PROGRAM EIP_COM
VAR
	eip_input AT%I* : ARRAY [0..63] OF BYTE;
	eip_output AT%Q* : ARRAY [0..63] OF BYTE;

END_VAR

eip_output := eip_input;

END_PROGRAM

(* stored: Version 1.1.0.1, ProductVersion 3.1.4024.12
   POU EIP_COM: Id {207ce353-6c4e-4027-a24a-2864afddaf38}, SpecialFunc None *)
